// Example of internal device communication.
FUNCTION_BLOCK FB_Ref_PubSub_Local EXTENDS FB_BA_View
VAR
	{region 'Analog'}
	
		A								: FB_BA_View := (
											iParent						:= THIS^,
											sDescription				:= '{Analog objects}'
										);
													 
			AV_Sub						: FB_BA_SubAPrio				:= (sSubject:='AV_Obj');
			AV_Obj						: FB_BA_AV := (
											iParent						:= A,
											iProfile					:= MyProfiles.AV_Prf,
											bEnPublish					:= TRUE
										); 
			AVOp_Sub					: FB_BA_SubAV_Op				:= (sSubject:='AVOp_Obj');
			AVOp_Obj					: FB_BA_AV_Op := (
											iParent						:= A,
											iProfile					:= MyProfiles.AVOp_Prf,
											bEnPublish					:= TRUE,
											fValueRm					:= 10
										); 
			AI_Sub						: FB_BA_SubAI					:= (sSubject:='AI_Obj');
			AI_Obj						: FB_BA_AI_Raw := (
											iParent						:= A,
											iProfile					:= MyProfiles.AI_Prf,
											bEnPublish					:= TRUE
										); 
			AO_Sub						: FB_BA_SubAPrio				:= (sSubject:='AO_Obj');
			AO_Obj						: FB_BA_AO_Raw := (
											iParent						:= A,
											iProfile					:= MyProfiles.AO_Prf,
											bEnPublish					:= TRUE
										); 
	{endregion}
	{region 'Binary'}
		B								: FB_BA_View := (
											iParent						:= THIS^,
											sDescription				:= '{Binary objects}'
										);
												 
			BV_Sub						: FB_BA_SubBPrio				:= (sSubject:='BV_Obj'); 
			BV_Obj						: FB_BA_BV := (
											iParent						:= B,
											iProfile					:= MyProfiles.BV_Prf,
											bEnPublish					:= TRUE
										);
			BVOp_Sub					: FB_BA_SubBV_Op				:= (sSubject:='BVOp_Obj');
			BVOp_Obj					: FB_BA_BV_Op := (
											iParent						:= B,
											iProfile					:= MyProfiles.BVOp_Prf,
											bEnPublish					:= TRUE,
											bValueRm					:= TRUE
										);
			BI_Sub						: FB_BA_SubBI					:= (sSubject:='BI_Obj');
			BI_Obj						: FB_BA_BI_Raw := (
											iParent						:= B,
											iProfile					:= MyProfiles.BI_Prf,
											bEnPublish					:= TRUE
										);
			BO_Sub						: FB_BA_SubBPrio				:= (sSubject:='BO_Obj');
			BO_Obj						: FB_BA_BO_Raw := (
											iParent						:= B,
											iProfile					:= MyProfiles.BO_Prf,
											bEnPublish					:= TRUE
										); 
	{endregion}
	{region 'Multistate'}
		M								: FB_BA_View := (
											iParent						:= THIS^,
											sDescription				:= '{Multistate objects}'
										);
			 
			MV_Sub						: FB_BA_SubMPrio				:= (sSubject:='MV_Obj');
			MV_Obj						: FB_BA_MV := (
											iParent						:= M,
											iProfile					:= MyProfiles.MV_Prf,
											bEnPublish					:= TRUE
										);
			MVOp_Sub					: FB_BA_SubMV_Op				:= (sSubject:='MVOp_Obj');
			MVOp_Obj					: FB_BA_MV_Op := (
											iParent						:= M,
											iProfile					:= MyProfiles.MVOp_Prf,
											bEnPublish					:= TRUE,
											nValueRm					:= 2
										);
			MI_Sub						: FB_BA_SubMI					:= (sSubject:='MI_Obj');
			MI_Obj						: FB_BA_MI_Raw := (
											iParent						:= M,
											iProfile					:= MyProfiles.MI_Prf,
											bEnPublish					:= TRUE
										);
			MO_Sub						: FB_BA_SubMPrio				:= (sSubject:='MO_Obj');
			MO_Obj						: FB_BA_MO_Raw := (
											iParent						:= M,
											iProfile					:= MyProfiles.MO_Prf,
											bEnPublish					:= TRUE
										); 
	{endregion}
	{region 'Multistate'}
		Misc							: FB_BA_View := (
											iParent						:= THIS^,
											sDescription				:= '{Miscellaneous objects}'
										);
			 
			Loop_Sub					: FB_BA_SubLoop					:= (sSubject:='Loop_Obj');
			Loop_Obj					: FB_BA_Loop := (
											iParent						:= Misc,
											iProfile					:= MyProfiles.Loop_Prf,
											bEnPublish					:= TRUE,
											fProportionalConstant		:= 5.0,
											fIntegralConstant			:= 180,
											bEn							:= TRUE,
											fSetpoint					:= 20,
											fCtrlVal					:= 25
										);
	                                    
			Cal_Sub						: FB_BA_SubCal					:= (sSubject:='Cal_Obj');
			Cal_Obj						: FB_BA_Cal := (
											iParent						:= Misc,
											iProfile					:= MyProfiles.Cal_Prf,
											bEnPublish					:= TRUE,
											aDateList := [(
												eType					:= E_BA_DateValChoice.eWeekNDay,
												uDate					:= F_BA_WeekNDayVal(E_BA_Weekday.eFriday, E_BA_Week.eWeek1, E_BA_Month.eFebruary)
											)]);
												 
			SchedA_Sub					: FB_BA_SubSchedA				:= (sSubject:='SchedA_Obj');
			SchedA_Obj					: FB_BA_SchedA := (
											iParent						:= Misc,
											iProfile					:= MyProfiles.SchedA_Prf,
											bEnPublish					:= TRUE,
											aWeek						:= F_BA_SchedWeekly3xA(E_BA_Weekday.eMonday, E_BA_Weekday.eFriday, T#0H, 0.0, T#6H, 5.0, T#20H, 0.0));
			SchedB_Sub					: FB_BA_SubSchedB				:= (sSubject:='SchedB_Obj');
			SchedB_Obj					: FB_BA_SchedB := (
											iParent						:= Misc,
											iProfile					:= MyProfiles.SchedB_Prf,
											bEnPublish					:= TRUE,
											aWeek						:= F_BA_SchedWeekly3xB(E_BA_Weekday.eMonday, E_BA_Weekday.eFriday, T#0H, FALSE, T#6H, TRUE, T#20H, FALSE));
			SchedM_Sub					: FB_BA_SubSchedM				:= (sSubject:='SchedM_Obj');
			SchedM_Obj					: FB_BA_SchedM := (
											iParent						:= Misc,
											iProfile					:= MyProfiles.SchedM_Prf,
											bEnPublish					:= TRUE,
											aWeek						:= F_BA_SchedWeekly3xM(E_BA_Weekday.eMonday, E_BA_Weekday.eFriday, T#0H, 1, T#6H, 2, T#20H, 1));
												 
			Trend_Sub					: FB_BA_SubTrend				:= (sSubject:='Trend_Obj');
			Trend_Obj					: FB_BA_Trend := (
											iParent						:= Misc,
											iProfile					:= MyProfiles.Trend_Prf,
											bEnPublish					:= TRUE,
											nEventClassID				:= 11,
											stReferredParam				:= F_BA_Reference(AV_Obj, E_BA_Parameter.ePresentValue)
										);
	{endregion}
	{region 'Custom'}
		{region 'Typed'}
			MyWthSt						: FB_BA_MyWeatherStation		:= (bEnPublish:= TRUE); 
			MyWthSt_Sub					: FB_BA_MyWeatherStationSub		:= (sSubject:='MyWthSt');
		{endregion}
		{region 'Raw'}
			MyRawWthStData				: ST_BA_MyWeatherData;
			MyRawWthSt					: FB_BA_RawPublisher;
					  
			MyRawWthStData_Sub			: ST_BA_MyWeatherData;
			MyRawWthSt_Sub				: FB_BA_RawSubscriber			:= (sSubject:='MyRawWthSt');
		{endregion}
	{endregion}
	{region 'Tests'}
		Tests							: FB_BA_View := (
											iParent						:= THIS^,
											sDescription				:= '{Test objects}'
										);
			 
		{region 'Subject path'}
			Nested1a					: FB_NestedView := (
											View						:= (iParent := Tests),
											Value						:= (bEnPublish := TRUE)
										);
			Nested1b					: FB_NestedView := (
											View						:= (iParent := Tests),
											Value						:= (bEnPublish := TRUE)
										);

			Nested1a_AV_Sub				: FB_BA_SubAV_Op := (
										//	sSubject					:= 'Val'							// -> Would lead to ambiguous subject!
											sSubject					:= 'Nested1a.Value'
										);
		{endregion}
	{endregion}
END_VAR

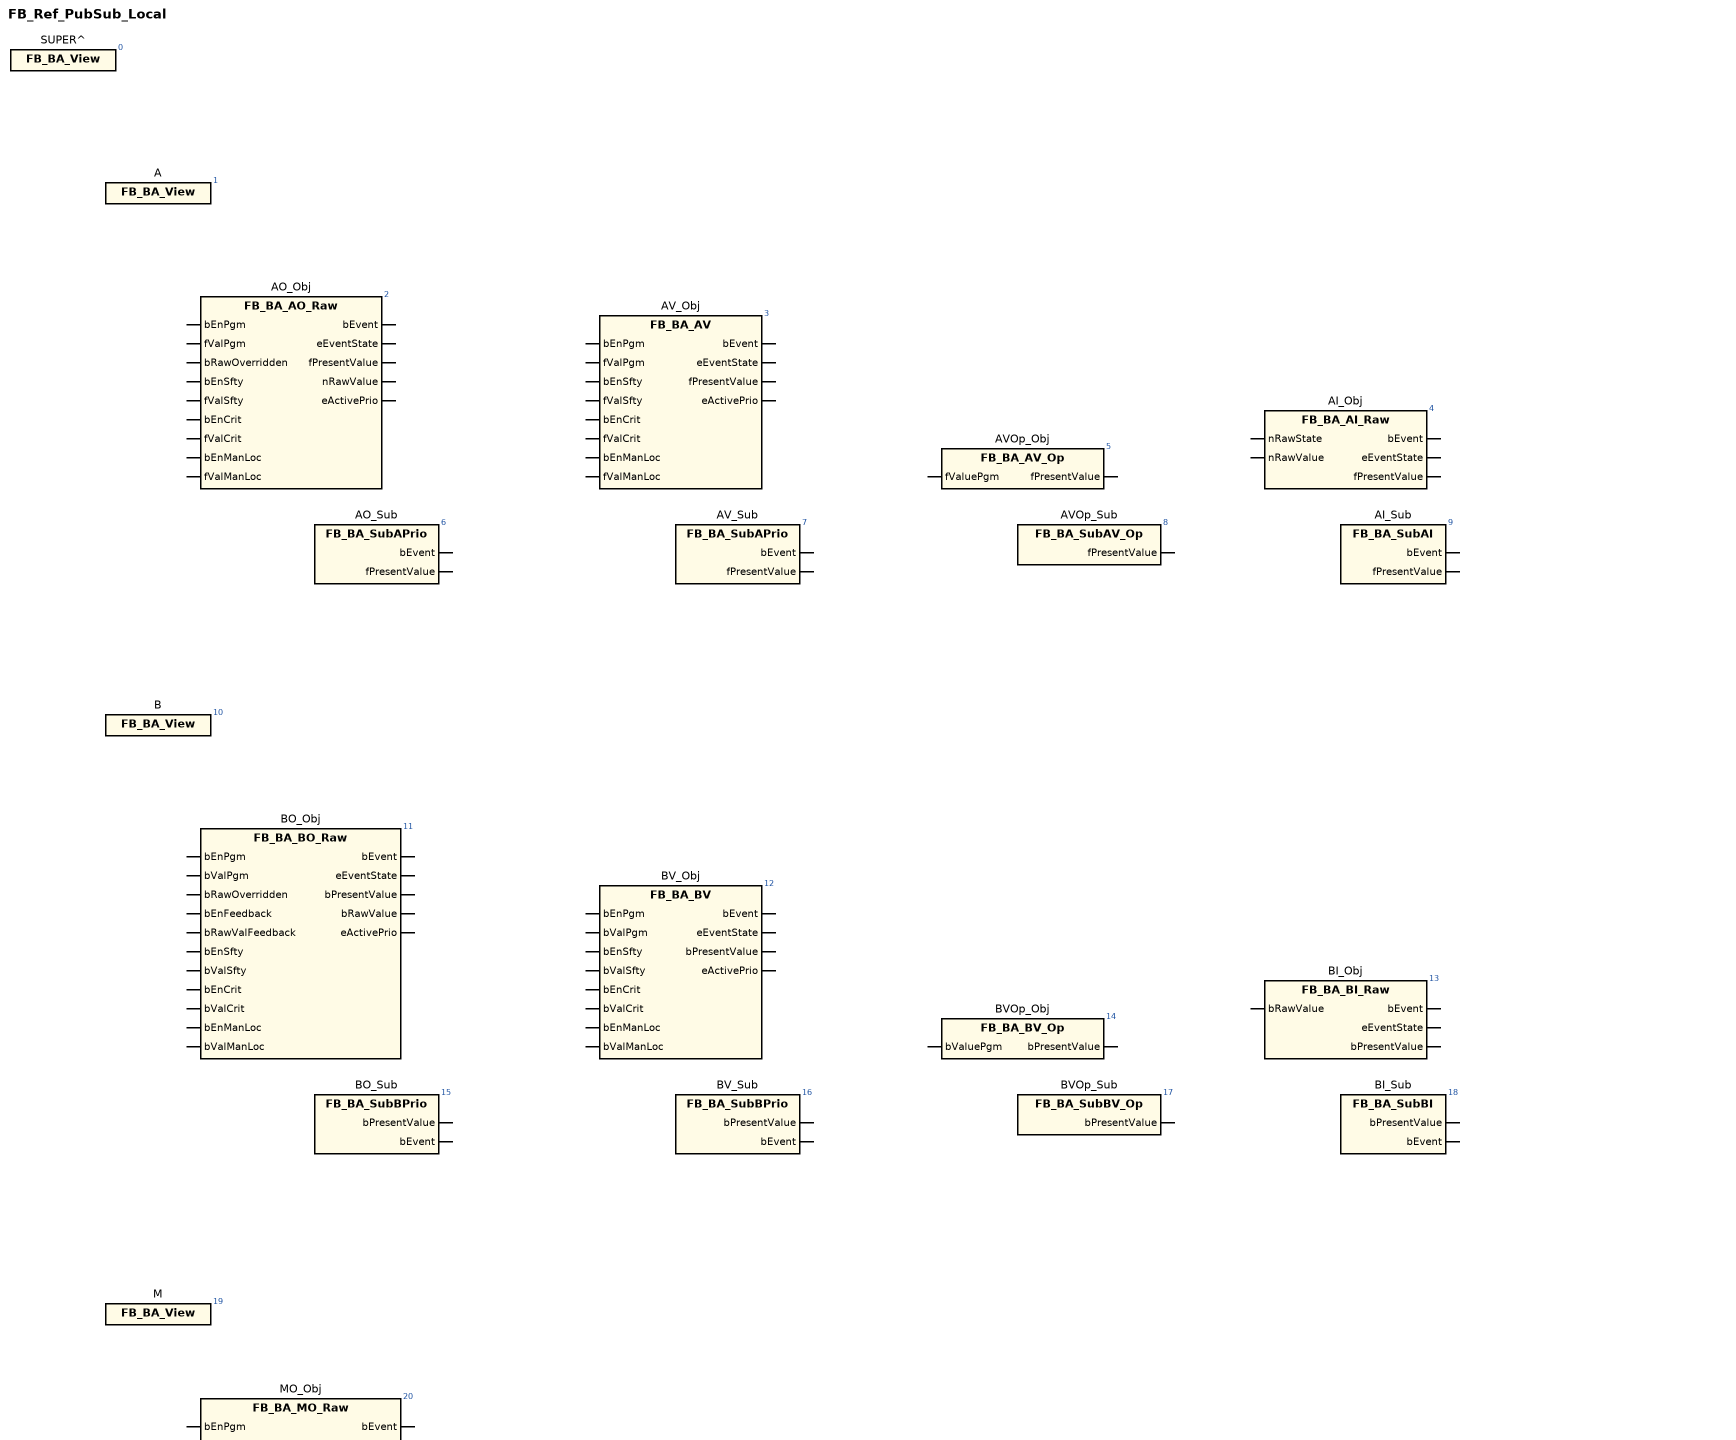
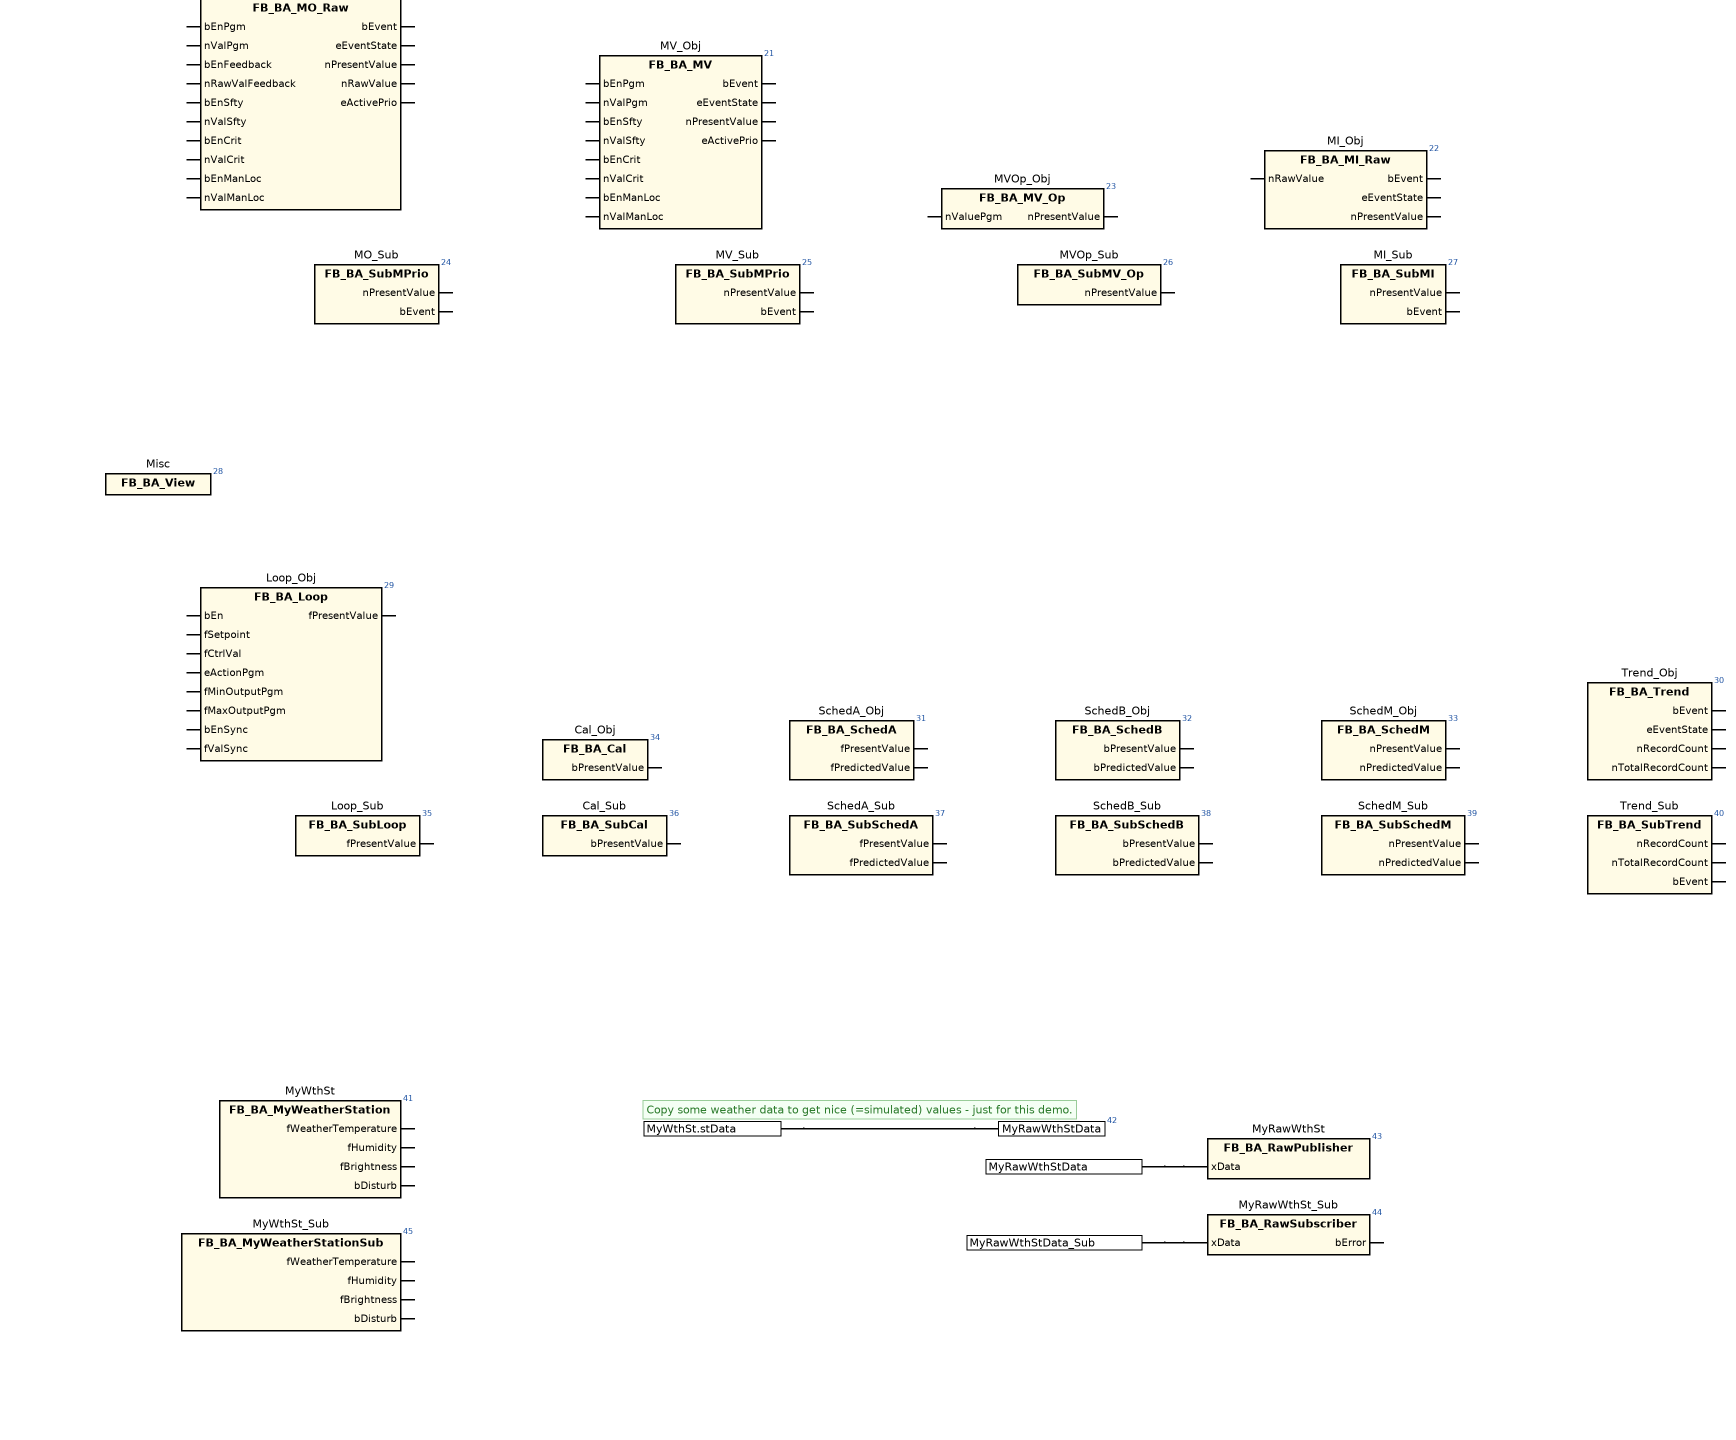
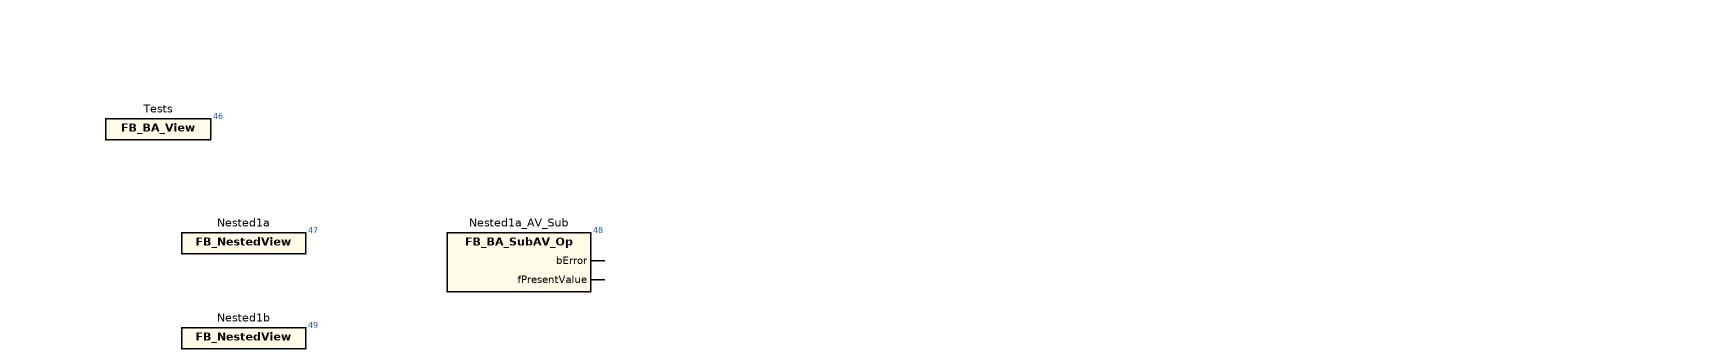
SUPER^(); // FB_BA_View
A(); // FB_BA_View
AO_Obj(); // FB_BA_AO_Raw
AV_Obj(); // FB_BA_AV
AI_Obj(); // FB_BA_AI_Raw
AVOp_Obj(); // FB_BA_AV_Op
AO_Sub(); // FB_BA_SubAPrio
AV_Sub(); // FB_BA_SubAPrio
AVOp_Sub(); // FB_BA_SubAV_Op
AI_Sub(); // FB_BA_SubAI
B(); // FB_BA_View
BO_Obj(); // FB_BA_BO_Raw
BV_Obj(); // FB_BA_BV
BI_Obj(); // FB_BA_BI_Raw
BVOp_Obj(); // FB_BA_BV_Op
BO_Sub(); // FB_BA_SubBPrio
BV_Sub(); // FB_BA_SubBPrio
BVOp_Sub(); // FB_BA_SubBV_Op
BI_Sub(); // FB_BA_SubBI
M(); // FB_BA_View
MO_Obj(); // FB_BA_MO_Raw
MV_Obj(); // FB_BA_MV
MI_Obj(); // FB_BA_MI_Raw
MVOp_Obj(); // FB_BA_MV_Op
MO_Sub(); // FB_BA_SubMPrio
MV_Sub(); // FB_BA_SubMPrio
MVOp_Sub(); // FB_BA_SubMV_Op
MI_Sub(); // FB_BA_SubMI
Misc(); // FB_BA_View
Loop_Obj(); // FB_BA_Loop
Trend_Obj(); // FB_BA_Trend
SchedA_Obj(); // FB_BA_SchedA
SchedB_Obj(); // FB_BA_SchedB
SchedM_Obj(); // FB_BA_SchedM
Cal_Obj(); // FB_BA_Cal
Loop_Sub(); // FB_BA_SubLoop
Cal_Sub(); // FB_BA_SubCal
SchedA_Sub(); // FB_BA_SubSchedA
SchedB_Sub(); // FB_BA_SubSchedB
SchedM_Sub(); // FB_BA_SubSchedM
Trend_Sub(); // FB_BA_SubTrend
MyWthSt(); // FB_BA_MyWeatherStation
// Copy some weather data to get nice (=simulated) values - just for this demo.
MyRawWthStData := MyWthSt.stData;
MyRawWthSt(xData := MyRawWthStData); // FB_BA_RawPublisher
MyRawWthSt_Sub(xData := MyRawWthStData_Sub); // FB_BA_RawSubscriber
MyWthSt_Sub(); // FB_BA_MyWeatherStationSub
Tests(); // FB_BA_View
Nested1a(); // FB_NestedView
Nested1a_AV_Sub(); // FB_BA_SubAV_Op
Nested1b(); // FB_NestedView

END_FUNCTION_BLOCK

(* stored: Version 1.1.0.1, ProductVersion 3.1.4024.5
   POU FB_Ref_PubSub_Local: Id {ef0e5899-b390-4c35-a440-3d3aad6b1c0b}, SpecialFunc None *)
